// TIA Portal V18 export
VAR_GLOBAL   // PLC tag table "Cabinet_7"
   Sz7_Button_LED_SS_Down AT %Q1700.0 : Bool;
   Sz7_Button_LED_SS_Up AT %Q1700.1 : Bool;
   Sz7_Button_LED_SS_Drive_ST35 AT %Q1700.2 : Bool;
   Sz7_Button_LED_SS_Drive_ST02 AT %Q1700.3 : Bool;
   Sz7_Button_LED_SS_Drive_ST03 AT %Q1700.4 : Bool;
   Sz7_Button_LED_SS_Drive_ST04 AT %Q1700.5 : Bool;
   Sz7_Button_LED_ST04_ST05 AT %Q1700.6 : Bool;
   Sz7_Button_LED_ST05_ST06 AT %Q1700.7 : Bool;
   "Reserved(76)" AT %Q1701.0 : Bool;
   "Reserved(77)" AT %Q1701.1 : Bool;
   "Reserved(78)" AT %Q1701.2 : Bool;
   "Reserved(79)" AT %Q1701.3 : Bool;
   "Reserved(80)" AT %Q1701.4 : Bool;
   "Reserved(81)" AT %Q1701.5 : Bool;
   "Reserved(82)" AT %Q1701.6 : Bool;
   "Reserved(83)" AT %Q1701.7 : Bool;
   Sz7_ST03_SenA AT %I1700.0 : Bool;
   Sz7_ST03_SenB AT %I1700.1 : Bool;
   Sz7_ST03_SenC AT %I1700.2 : Bool;
   Sz7_ST03_SenD AT %I1700.3 : Bool;
   Sz7_ST04_SenA AT %I1700.4 : Bool;
   Sz7_ST04_SenB AT %I1700.5 : Bool;
   Sz7_ST04_SenC AT %I1700.6 : Bool;
   Sz7_ST04_SenD AT %I1700.7 : Bool;
   Sz7_ST04_SenE AT %I1701.0 : Bool;
   Sz7_ST04_SenF AT %I1701.1 : Bool;
   Sz7_ST05_SenA AT %I1701.2 : Bool;
   Sz7_ST05_SenB AT %I1701.3 : Bool;
   Sz7_ST05_SenC AT %I1701.4 : Bool;
   Sz7_ST05_SenD AT %I1701.5 : Bool;
   "Reserved(84)" AT %I1701.6 : Bool;
   "Reserved(85)" AT %I1701.7 : Bool;
   Sz7_Button_SS_Down AT %I1702.0 : Bool;
   Sz7_Safety1_1 AT %I1750.0 : Bool;
   Sz7_Button_SS_Up AT %I1702.1 : Bool;
   Sz7_Button_SS_Drive_ST35 AT %I1702.2 : Bool;
   Sz7_Button_SS_Drive_ST02 AT %I1702.3 : Bool;
   Sz7_Button_SS_Drive_ST03 AT %I1702.4 : Bool;
   Sz7_Button_SS_Drive_ST04 AT %I1702.5 : Bool;
   Sz7_Button_ST04_ST05 AT %I1702.6 : Bool;
   Sz7_Button_ST05_ST06 AT %I1702.7 : Bool;
   "Reserved(100)" AT %I1703.0 : Bool;
   "Reserved(101)" AT %I1703.1 : Bool;
   "Reserved(102)" AT %I1703.2 : Bool;
   "Reserved(103)" AT %I1703.3 : Bool;
   "Reserved(104)" AT %I1703.4 : Bool;
   "Reserved(105)" AT %I1703.5 : Bool;
   "Reserved(106)" AT %I1703.6 : Bool;
   "Reserved(107)" AT %I1703.7 : Bool;
   "Reserved(86)" AT %I1750.1 : Bool;
   "Reserved(87)" AT %I1750.2 : Bool;
   "Reserved(88)" AT %I1750.3 : Bool;
   "Sz7-Safety1_2" AT %I1750.4 : Bool;
   "Reserved(89)" AT %I1750.5 : Bool;
   "Reserved(90)" AT %I1750.6 : Bool;
   "Reserved(91)" AT %I1750.7 : Bool;
   "Reserved(92)" AT %I1751.0 : Bool;
   "Reserved(93)" AT %I1751.1 : Bool;
   "Reserved(94)" AT %I1751.2 : Bool;
   "Reserved(95)" AT %I1751.3 : Bool;
   "Reserved(96)" AT %I1751.4 : Bool;
   "Reserved(97)" AT %I1751.5 : Bool;
   "Reserved(98)" AT %I1751.6 : Bool;
   "Reserved(99)" AT %I1751.7 : Bool;
END_VAR
